TYPE STATE:
    STRUCT
        curTime: REAL;
        dvar_M_aut_y: DINT;
    END_STRUCT;
END_TYPE
